Fanuc KAREL source: ko00074.KL

-- PROVISIONAL review KL for V770-1; original PC SHA256 2b3ed091d00c3c8206e0a8147b854771e1d8582eeb500a24948f759394d46e74
-- Incomplete behavior may be omitted. Consult companion uncertainty JSON. Do not deploy.
PROGRAM KO00074
%NOLOCKGROUP
BEGIN
  -- UNRESOLVED_PC offsets 5-12; opcodes 9D,23
  -- UNRESOLVED_PC offsets 17-66; opcodes 27,22,1C,27,49,7E,AD,22,31,7E,4A
  -- UNRESOLVED_PC offsets 71-75; opcodes 7F
END KO00074
